// TIA Portal V18 export
// export: Created 2025-12-01T17:51:15.217276Z, ExportSetting None, DisplayName Totally Integrated Automation Portal, DisplayVersion V18 Update 5, DisplayName TIA Portal Openness, DisplayVersion V18 Update 5, DisplayName TIA Portal Teamcenter Gateway, DisplayVersion V18, DisplayName TIA Portal Version Control Interface, DisplayVersion V18, DisplayName STEP 7 Professional, DisplayVersion V18 Update 5, DisplayName STEP 7 Safety, DisplayVersion V18, DisplayName WinCC Professional, DisplayVersion V18 Update 5
DATA_BLOCK "KukaRobot3_CtrlDB"   // DB2403
// stored: AutoNumber false, InstanceOfName KukaRobot3_Ctrl, InstanceOfType FB
"KukaRobot3_Ctrl"
   // VAR_INPUT
   //    iHWID_In : HW_IO;
   //    iHWID_Out : HW_IO;
   //    iSysRun : Bool;
   //    iAuto : Bool;
   //    iManual : Bool;
   //    iSpecial : Bool;
   //    iE_STOP : Bool;
   //    iReset : Bool;
   //    iT1000ms : Bool;
   //    iTaskMode : USInt;
   //    iPartType : USInt;
   //    iSpeedValue : USInt;
   //    iPGNO : USInt;
   // END_VAR
   // VAR_OUTPUT
   //    oReady : Bool;
   //    oStartComplete : Bool;
   //    oWarning : Bool;
   //    oError : Bool;
   //    oErrorCode : Int;
   // END_VAR
   // VAR_IN_OUT
   //    ioAutoStart : Bool;
   //    ioSrartHome : Bool;
   //    ioStartAutoCycle : Bool;
   // END_VAR
   // VAR RETAIN
   //    sHMI { S7_SetPoint := 'True'} : "KukaRobot_HMI";
   //    sROBtoPLC : Struct
   //       Sys { S7_SetPoint := 'True'} : "KukaRobot_SysOutput";
   //       User { S7_SetPoint := 'True'} : "KukaRobot_UserOutput_3";
   //    END_STRUCT;
   //    sPLCtoROB : Struct
   //       Sys { S7_SetPoint := 'True'} : "KukaRobot_SysInput";
   //       User { S7_SetPoint := 'True'} : "KukaRobot_UserInput_3";
   //    END_STRUCT;
   //    sDrivesOnDelay { S7_SetPoint := 'True'} : TON_TIME;
   //    sStartUpDelay { S7_SetPoint := 'True'} : TON_TIME;
   //    sRobotReadyToStart : Bool;
   //    sRobotReadyToRunning : Bool;
   //    sRobotActComplete : Bool;
   //    sRobotProgrameChoseOK : Bool;
   //    sSequence : Int;
   //    F_TRIG_Work { S7_SetPoint := 'True'} : F_TRIG;
   //    F_TRIG_Home { S7_SetPoint := 'True'} : F_TRIG;
   //    ModeValue : Int;
   //    Tem_ModeValue : Int;
   //    ModeChange : Bool;
   //    IEC_Timer_DRIVES_OFF { S7_SetPoint := 'True'} : TON_TIME;
   //    IEC_Timer_DRIVES_ON { S7_SetPoint := 'True'} : TON_TIME;
   // END_VAR
BEGIN
   // sROBtoPLC.User.Safety.DO450 : BRAKETEST_MONTIME
   // sROBtoPLC.User.Safety.DO451 : MAINTENANCE_TO_PLC
   // sROBtoPLC.User.Safety.DO452 : BRAKETEST_REQ_INT
   // sROBtoPLC.User.Safety.DO453 : BRAKETEST_WORK
   // sROBtoPLC.User.Safety.DO454 : BRAKES_OK
   // sROBtoPLC.User.Safety.DO455 : BRAKETEST_WARN
   // sROBtoPLC.User.Safety.DO456 : SPOC_MOTION_ENABLE
   // sROBtoPLC.User.Safety.DO457 : COLLISION
   // sROBtoPLC.User.Safety.DO458 : COLLISION_STOP
   // sROBtoPLC.User.Safety.DO460 : MASTERINGTEST_REQ_INT
   // sROBtoPLC.User.Safety.DO461 : MASTERINGTEST_SWITCH_ OK
   // sROBtoPLC.User.Safety.DO462 : MASTERINGTEST_ACTIVE
   // sPLCtoROB.User.Home.DI170 : Robot 2 safe area
   // sPLCtoROB.User.Cycle.DI321 : MASTERINGTEST_REQ_INT
   // sPLCtoROB.User.Cycle.DI329 : BRAKETEST_REQ_INT
END_DATA_BLOCK
